(* PLC project control_valve, Dassault Systèmes ControlBuild 2024x *)
(* stored: creationDateTime 2023-10-03T11:12:59-01:00 *)

(* This module simulates the behaviour of a control valve and its electrical control logic. *)
FUNCTION_BLOCK equipment_library.control_valve
  VAR_INPUT
    inputFlow : REAL := 0.0;
  END_VAR
  VAR_INPUT
    voltage380 : BOOL := true;
    cmdSupply : BOOL := true;
    sensorSupply : BOOL := true;
  END_VAR
  VAR_INPUT
    onCmd : BOOL := false;
    setpoint : REAL := 0.0;
  END_VAR
  VAR_OUTPUT
    openedSensor : BOOL := false;
    closedSensor : BOOL := false;
  END_VAR
  VAR_OUTPUT
    outputFlow : REAL := 0.0;
    percentOpening : REAL := 0.0;
  END_VAR
  VAR
    increment : REAL := 0.0;
    openingVal : REAL := 0.0;
    unit : REAL := 0.0;
  END_VAR
  VAR CONSTANT
    openingTime : DINT := 2;
    flowMax : REAL := 10000.0;
    openedSensorLogic : BOOL := true;
    closedSensorLogic : BOOL := true;
    flowPerHour : BOOL := true;
    flowPerMinute : BOOL := false;
  END_VAR
  VAR
    d_locking : BOOL := false;
    v_d_locking : REAL := 0.0;
    d_flow : BOOL := false;
    v_d_flow : REAL := 0.0;
    d_electrical : BOOL := false;
    v_d_electrical : BOOL := false;
    d_closedSensor : BOOL := false;
    v_d_closedSensor : BOOL := false;
    d_openedSensor : BOOL := false;
    v_d_openedSensor : BOOL := false;
  END_VAR


ACTION C_source_code:
/* -----------------------------------------------------------------	*/
/* Type : Model of Operative Behaviour					*/
/* Catégorie :   batch							*/
/* Author : Dassault Systemes						*/
/* Update date : June 2018							*/
/* -----------------------------------------------------------------	*/
/* This module simulates the behaviour of a control valve and its	*/
/* electrical control logic.						*/
/* The setpoint can go from 0% up to +100%.				*/
/* ----------------------------------------------------------------	*/

/* ----------------------------------------------------------------	*/
/* Management of opening							*/
/* ----------------------------------------------------------------	*/
if (( ! d_locking) && (voltage380) && (! d_electrical) && (cmdSupply) && (onCmd)) {

	/* Compute the increment of opening according to the simulation clock	*/
	if (openingTime > 0.0)
		increment = (100.0  / openingTime) * (CLOCK_PERIOD/1000000);

	/* Compute the opening	*/
	if ((openingVal < fabs(setpoint))  &&  (fabs(setpoint) <= 100.0)) {
		(openingVal) += increment;
		if (openingVal > fabs(setpoint)) openingVal = fabs(setpoint);
	}

	if (openingVal > fabs(setpoint)) {
		(openingVal) -= increment;
		if (openingVal < fabs(setpoint)) openingVal = fabs(setpoint);
		if (openingVal < 0.0) openingVal = 0.0;
	}
}

if (d_locking)
	openingVal = v_d_locking;

/* ----------------------------------------------------------------	*/
/* Compute the percentage of opening					*/
/* ----------------------------------------------------------------	*/
percentOpening = ((openingVal / 100.0) * 100.0);

/* ----------------------------------------------------------------	*/
/* Management of flow rate 	 						*/
/* ----------------------------------------------------------------	*/
if (d_flow)
	outputFlow = v_d_flow;
else {
	if (flowPerHour) unit = 3600.0;
	else if (flowPerMinute) unit = 60.0;
		else unit = 1.0;
	
	outputFlow = ((flowMax * CLOCK_PERIOD / 1000000)  / unit) * (percentOpening  /100.0);
	if (outputFlow > inputFlow) outputFlow = inputFlow;
		
}

/* ----------------------------------------------------------------	*/
/* Management of sensors' state						*/
/* ----------------------------------------------------------------	*/
if (d_openedSensor) openedSensor = v_d_openedSensor;
else
	openedSensor = ((openingVal >= 100.0) ^ ! openedSensorLogic) && sensorSupply;

if (d_closedSensor) closedSensor = v_d_closedSensor;
else
	closedSensor = ((openingVal == 0.0) ^ ! closedSensorLogic) && sensorSupply;
END_ACTION

ACTION C_header:
#include <math.h>
END_ACTION
END_FUNCTION_BLOCK
